// TIA Portal V21 export
FUNCTION_BLOCK "TIME_COUNTER_FB"   // FB9000, LAD
{ S7_Optimized_Access := 'TRUE' }
// TIME COUNTER [S, M, H]
// stored: AutoNumber false, MemoryReserve 100, SetENOAutomatically false
   VAR_INPUT
      FI_START_COUNTING : Bool;
   END_VAR
   VAR_IN_OUT
      FIQ_TIMER : "UDT_WORK_CNT";
   END_VAR
   VAR
      E1 : Bool;
      E2 : Bool;
      RESET_CTU : Bool;
   END_VAR
   VAR_TEMP   // added for the SCL form of the ladder/FBD networks
      _w1 : Bool;
   END_VAR
BEGIN

REGION Network 1: COUNTERS INCREMENT
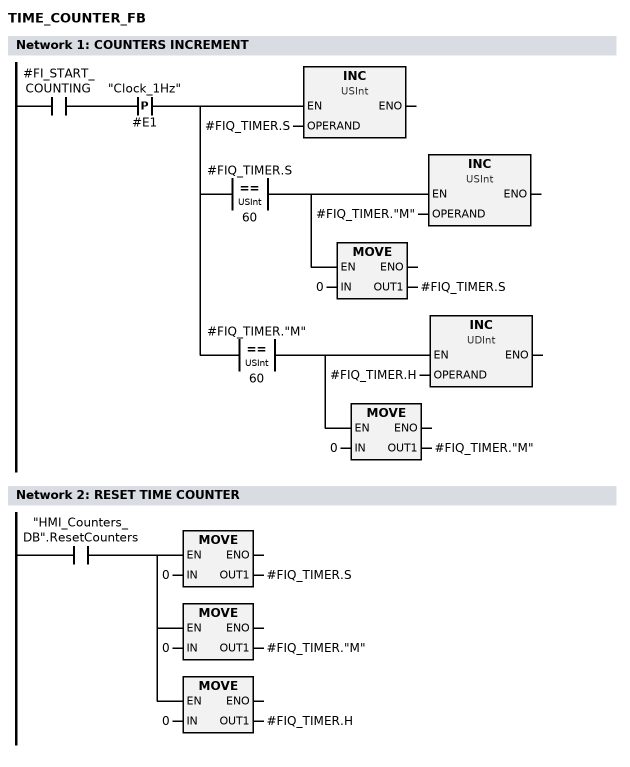
   RUNG wire#powerrail
      Contact( #FI_START_COUNTING )
      P_Contact(operand := "Clock_1Hz", bit := #E1)
      wire#w1
      { S7_Templates := "DestType := USInt" } Inc( #FIQ_TIMER.S )
   END_RUNG
   RUNG wire#w1
      { S7_Templates := "SrcType := USInt" } EQ_Contact(in1 := #FIQ_TIMER.S, in2 := 60)
      wire#w2
      { S7_Templates := "DestType := USInt" } Inc( #FIQ_TIMER."M" )
   END_RUNG
   RUNG wire#w2
      Move(in := 0, out1 => #FIQ_TIMER.S)
   END_RUNG
   RUNG wire#w1
      { S7_Templates := "SrcType := USInt" } EQ_Contact(in1 := #FIQ_TIMER."M", in2 := 60)
      wire#w3
      { S7_Templates := "DestType := UDInt" } Inc( #FIQ_TIMER.H )
   END_RUNG
   RUNG wire#w3
      Move(in := 0, out1 => #FIQ_TIMER."M")
   END_RUNG
   // the same network as SCL:
   #_w1 := #FI_START_COUNTING AND "Clock_1Hz" AND NOT #E1;   // rising edge of "Clock_1Hz"
   #E1 := "Clock_1Hz";
   IF #_w1 THEN #FIQ_TIMER.S := #FIQ_TIMER.S + 1; END_IF;
   IF #_w1 AND (#FIQ_TIMER.S = 60) THEN
       #FIQ_TIMER."M" := #FIQ_TIMER."M" + 1;
       #FIQ_TIMER.S := 0;
   END_IF;
   IF #_w1 AND (#FIQ_TIMER."M" = 60) THEN
       #FIQ_TIMER.H := #FIQ_TIMER.H + 1;
       #FIQ_TIMER."M" := 0;
   END_IF;
END_REGION

REGION Network 2: RESET TIME COUNTER
   RUNG wire#powerrail
      Contact( "HMI_Counters_DB".ResetCounters )
      wire#w1
      Move(in := 0, out1 => #FIQ_TIMER.S)
   END_RUNG
   RUNG wire#w1
      Move(in := 0, out1 => #FIQ_TIMER."M")
   END_RUNG
   RUNG wire#w1
      Move(in := 0, out1 => #FIQ_TIMER.H)
   END_RUNG
   // the same network as SCL:
   IF "HMI_Counters_DB".ResetCounters THEN
       #FIQ_TIMER.S := 0;
       #FIQ_TIMER."M" := 0;
       #FIQ_TIMER.H := 0;
   END_IF;
END_REGION
END_FUNCTION_BLOCK
